Staubli VAL3: IO123.dtx

mdesc mNomSpeed
public string sIOName
public bool bDigtal
